# EPICS autosave request: apps/plcApp/Db/HPS_SVT_Interlocks.req
file HPS_SVT_Interlock_v5_PLC.req IOC=${PREF}:i
file HPS_SVT_Interlock_v5_PLC.req IOC=${PREF}:o
